{attribute 'GeneratedUsingTerminal: EL3423-0000-0016'}
{attribute addProperty BoxType "EL3423-0000-0016"}
{attribute addProperty Id "Reset_IntervalAT %Q*BOOL1"}
{attribute addProperty CRC "360233940"}
{attribute addProperty Size "1"}
TYPE Interval_1578BBD4 EXTENDS OutputBase_10CEE7DE :
STRUCT
	{attribute addProperty Name "Reset_Interval"}
	Reset_Interval AT %Q* : BOOL;
END_STRUCT
END_TYPE

(* stored: Version 1.2.0.0, ProductVersion 3.1.4024.9
   DUT Interval_1578BBD4: Id {0a5280df-81a7-477f-8ee9-463fdb13f5e7} *)
